Staubli VAL3: Carterblend.pgx

program Carterblend()
begin

  //直线与圆弧



  //直线与直线




  //圆弧与直线



  //圆弧与圆弧














end
